    // Motor axes
    {attribute 'pytmc' := 'pv: CRIX:DPL:MMS:X'}
    {attribute 'TcLinkTo' := '.bLimitForwardEnable  := TIID^Device 1 (EtherCAT)^Term 5 (EK1200)^Term 6 (EK1122-0080)^DRL02-EK0 (EK1101-0080)^DRL02-E1 (EL7031)^STM Status^Status^Digital input 2;
                              .bLimitBackwardEnable := TIID^Device 1 (EtherCAT)^Term 5 (EK1200)^Term 6 (EK1122-0080)^DRL02-EK0 (EK1101-0080)^DRL02-E1 (EL7031)^STM Status^Status^Digital input 1'}
    M1 : DUT_MotionStage := (bPowerSelf:=TRUE, nEnableMode:=ENUM_StageEnableMode.DURING_MOTION);
    //stDPXMotor : DUT_MotionStage;

    {attribute 'pytmc' := 'pv: CRIX:DPL:MMS:Y'}
    {attribute 'TcLinkTo' := '.bLimitForwardEnable  := TIID^Device 1 (EtherCAT)^Term 5 (EK1200)^Term 6 (EK1122-0080)^DRL02-EK0 (EK1101-0080)^DRL02-E3 (EL7031)^STM Status^Status^Digital input 1;
                              .bLimitBackwardEnable := TIID^Device 1 (EtherCAT)^Term 5 (EK1200)^Term 6 (EK1122-0080)^DRL02-EK0 (EK1101-0080)^DRL02-E3 (EL7031)^STM Status^Status^Digital input 2'}
    M2 : DUT_MotionStage := (bPowerSelf:=TRUE, nEnableMode:=ENUM_StageEnableMode.DURING_MOTION);
    //stDPYMotor : DUT_MotionStage;

    {attribute 'pytmc' := 'pv: CRIX:DPL:MMS:Z'}
    {attribute 'TcLinkTo' := '.bLimitForwardEnable  := TIID^Device 1 (EtherCAT)^Term 5 (EK1200)^Term 6 (EK1122-0080)^DRL02-EK0 (EK1101-0080)^DRL02-E4 (EL7031)^STM Status^Status^Digital input 1;
                              .bLimitBackwardEnable := TIID^Device 1 (EtherCAT)^Term 5 (EK1200)^Term 6 (EK1122-0080)^DRL02-EK0 (EK1101-0080)^DRL02-E4 (EL7031)^STM Status^Status^Digital input 2'}
    M3 : DUT_MotionStage :=(bPowerSelf:=TRUE,nEnableMode:=ENUM_StageEnableMode.DURING_MOTION);
    //stDPZMotor : DUT_MotionStage;




    {attribute 'pytmc' := 'pv: CRIX:OBJ:MMS:X'}
    {attribute 'TcLinkTo' := '.bLimitForwardEnable  := TIID^Device 1 (EtherCAT)^Term 5 (EK1200)^Term 6 (EK1122-0080)^DRL02-EK0 (EK1101-0080)^DRL02-E6 (EL7031)^STM Status^Status^Digital input 2;
                              .bLimitBackwardEnable := TIID^Device 1 (EtherCAT)^Term 5 (EK1200)^Term 6 (EK1122-0080)^DRL02-EK0 (EK1101-0080)^DRL02-E6 (EL7031)^STM Status^Status^Digital input 1'}
    M4: DUT_MotionStage :=(bPowerSelf:=TRUE ,nEnableMode:=ENUM_StageEnableMode.DURING_MOTION);
    //stOBJXMotor : DUT_MotionStage;

    {attribute 'pytmc' := 'pv: CRIX:OBJ:MMS:Y'}
    {attribute 'TcLinkTo' := '.bLimitForwardEnable  := TIID^Device 1 (EtherCAT)^Term 5 (EK1200)^Term 6 (EK1122-0080)^DRL02-EK0 (EK1101-0080)^DRL02-E7 (EL7031)^STM Status^Status^Digital input 1;
                              .bLimitBackwardEnable := TIID^Device 1 (EtherCAT)^Term 5 (EK1200)^Term 6 (EK1122-0080)^DRL02-EK0 (EK1101-0080)^DRL02-E7 (EL7031)^STM Status^Status^Digital input 2'}
    M5 : DUT_MotionStage :=(bPowerSelf:=TRUE, nEnableMode:=ENUM_StageEnableMode.DURING_MOTION);
    //stOBJYMotor : DUT_MotionStage;

    {attribute 'pytmc' := 'pv: CRIX:OBJ:MMS:Z'}
    {attribute 'TcLinkTo' := '.bLimitForwardEnable  := TIID^Device 1 (EtherCAT)^Term 5 (EK1200)^Term 6 (EK1122-0080)^DRL02-EK0 (EK1101-0080)^DRL02-E9 (EL7031)^STM Status^Status^Digital input 1;
                              .bLimitBackwardEnable := TIID^Device 1 (EtherCAT)^Term 5 (EK1200)^Term 6 (EK1122-0080)^DRL02-EK0 (EK1101-0080)^DRL02-E9 (EL7031)^STM Status^Status^Digital input 2'}
    M6 : DUT_MotionStage :=(bPowerSelf:=TRUE, nEnableMode:=ENUM_StageEnableMode.DURING_MOTION);
    //stOBJZMotor : DUT_MotionStage;



    {attribute 'pytmc' := 'pv: CRIX:PDET:MMS:Y'}
    {attribute 'TcLinkTo' := '.bLimitForwardEnable  := TIID^Device 1 (EtherCAT)^Term 5 (EK1200)^Term 6 (EK1122-0080)^DRL02-EK0 (EK1101-0080)^DRL02-E11 (EL7031)^STM Status^Status^Digital input 1;
                              .bLimitBackwardEnable := TIID^Device 1 (EtherCAT)^Term 5 (EK1200)^Term 6 (EK1122-0080)^DRL02-EK0 (EK1101-0080)^DRL02-E11 (EL7031)^STM Status^Status^Digital input 2'}
    M7 : DUT_MotionStage := (bPowerSelf:=TRUE, nEnableMode:=ENUM_StageEnableMode.DURING_MOTION);
    //stPDYMotor : DUT_MotionStage;
    {attribute 'pytmc' := 'pv: CRIX:PDET:MMS:THETA'}
    {attribute 'TcLinkTo' := '.bLimitForwardEnable  := TIID^Device 1 (EtherCAT)^Term 5 (EK1200)^Term 6 (EK1122-0080)^DRL02-EK0 (EK1101-0080)^DRL02-E13 (EL7041)^STM Status^Status^Digital input 1;
                              .bLimitBackwardEnable := TIID^Device 1 (EtherCAT)^Term 5 (EK1200)^Term 6 (EK1122-0080)^DRL02-EK0 (EK1101-0080)^DRL02-E13 (EL7041)^STM Status^Status^Digital input 2'}
    M8 : DUT_MotionStage := (bPowerSelf:=TRUE, nEnableMode:=ENUM_StageEnableMode.DURING_MOTION);
    //stPDRotMotor : DUT_MotionStage;

    {attribute 'pytmc' := 'pv: CRIX:ILM:MMS:X'}
    {attribute 'TcLinkTo' := '.bLimitForwardEnable  := TIID^Device 1 (EtherCAT)^Term 5 (EK1200)^Term 6 (EK1122-0080)^DRL02-EK0 (EK1101-0080)^Term 65 (EL1084)^Channel 1^Input;
                              .bLimitBackwardEnable := TIID^Device 1 (EtherCAT)^Term 5 (EK1200)^Term 6 (EK1122-0080)^DRL02-EK0 (EK1101-0080)^Term 65 (EL1084)^Channel 2^Input'}
    M9 : DUT_MotionStage := (bPowerSelf:=TRUE, nEnableMode:=ENUM_StageEnableMode.DURING_MOTION); //stILMXMotor : DUT_MotionStage;

    {attribute 'pytmc' := 'pv: CRIX:ILM:MMS:Y'}
    {attribute 'TcLinkTo' := '.bLimitForwardEnable  := TIID^Device 1 (EtherCAT)^Term 5 (EK1200)^Term 6 (EK1122-0080)^DRL02-EK0 (EK1101-0080)^Term 65 (EL1084)^Channel 3^Input;
                              .bLimitBackwardEnable := TIID^Device 1 (EtherCAT)^Term 5 (EK1200)^Term 6 (EK1122-0080)^DRL02-EK0 (EK1101-0080)^Term 65 (EL1084)^Channel 4^Input'}
    M10 : DUT_MotionStage := (bPowerSelf:=TRUE, nEnableMode:=ENUM_StageEnableMode.DURING_MOTION); //stILMYMotor : DUT_MotionStage;

    {attribute 'pytmc' := 'pv: CRIX:ILM:MMS:Z'}
    {attribute 'TcLinkTo' := '.bLimitForwardEnable  := TIID^Device 1 (EtherCAT)^Term 5 (EK1200)^Term 6 (EK1122-0080)^DRL02-EK0 (EK1101-0080)^Term 68 (EL1084)^Channel 1^Input;
                              .bLimitBackwardEnable := TIID^Device 1 (EtherCAT)^Term 5 (EK1200)^Term 6 (EK1122-0080)^DRL02-EK0 (EK1101-0080)^Term 68 (EL1084)^Channel 2^Input'}
    M11 : DUT_MotionStage := (bPowerSelf:=TRUE, nEnableMode:=ENUM_StageEnableMode.DURING_MOTION); //stILMZMotor : DUT_MotionStage;

    {attribute 'pytmc' := 'pv: CRIX:QSTR:MMS:X'}
    {attribute 'TcLinkTo' := '.bLimitForwardEnable  := TIID^Device 1 (EtherCAT)^Term 5 (EK1200)^Term 6 (EK1122-0080)^DRL02-EK0 (EK1101-0080)^DRL02-E17 (EL7031)^STM Status^Status^Digital input 1;
                              .bLimitBackwardEnable := TIID^Device 1 (EtherCAT)^Term 5 (EK1200)^Term 6 (EK1122-0080)^DRL02-EK0 (EK1101-0080)^DRL02-E17 (EL7031)^STM Status^Status^Digital input 2'}
    M12 : DUT_MotionStage := (bPowerSelf:=TRUE, nEnableMode:=ENUM_StageEnableMode.DURING_MOTION);
    //stQSTXMotor : DUT_MotionStage;
    {attribute 'pytmc' := 'pv: CRIX:QSTR:MMS:Y'}
    {attribute 'TcLinkTo' := '.bLimitForwardEnable  := TIID^Device 1 (EtherCAT)^Term 5 (EK1200)^Term 6 (EK1122-0080)^DRL02-EK0 (EK1101-0080)^DRL02-E19 (EL7031)^STM Status^Status^Digital input 1;
                              .bLimitBackwardEnable := TIID^Device 1 (EtherCAT)^Term 5 (EK1200)^Term 6 (EK1122-0080)^DRL02-EK0 (EK1101-0080)^DRL02-E19 (EL7031)^STM Status^Status^Digital input 2'}
    M13 : DUT_MotionStage := (bPowerSelf:=TRUE, nEnableMode:=ENUM_StageEnableMode.DURING_MOTION);
    //stQSTYMotor : DUT_MotionStage;

    M14 : DUT_MotionStage; // SPARE 1
    M15 : DUT_MotionStage; // SPARE 2

    {attribute 'pytmc' := 'pv: CRIX:SDS:MMS:X'}
    M16 : DUT_MotionStage := (bPowerSelf:=TRUE, nEnableMode:=ENUM_StageEnableMode.DURING_MOTION); //stSDSXMotor : DUT_MotionStage;

    {attribute 'pytmc' := 'pv: CRIX:SDS:MMS:Y'}
    {attribute 'TcLinkTo' := '.bLimitForwardEnable := TIID^Device 1 (EtherCAT)^Term 5 (EK1200)^Term 6 (EK1122-0080)^DRL02-EK0 (EK1101-0080)^DRL02-E26 (EL7031)^STM Status^Status^Digital input 1;
                              .bLimitBackwardEnable := TIID^Device 1 (EtherCAT)^Term 5 (EK1200)^Term 6 (EK1122-0080)^DRL02-EK0 (EK1101-0080)^DRL02-E26 (EL7031)^STM Status^Status^Digital input 2'}
    M17 : DUT_MotionStage := (bPowerSelf:=TRUE, nEnableMode:=ENUM_StageEnableMode.DURING_MOTION); //stSDSYMotor : DUT_MotionStage;

    {attribute 'pytmc' := 'pv: CRIX:SDS:MMS:Z'}
    {attribute 'TcLinkTo' := '.bLimitForwardEnable := TIID^Device 1 (EtherCAT)^Term 5 (EK1200)^Term 6 (EK1122-0080)^DRL02-EK0 (EK1101-0080)^DRL02-E27 (EL7031)^STM Status^Status^Digital input 1'}
    M18 : DUT_MotionStage := (bPowerSelf:=TRUE, nEnableMode:=ENUM_StageEnableMode.DURING_MOTION); //stSDSZMotor : DUT_MotionStage;

    {attribute 'pytmc' := 'pv: CRIX:SDS:MMS:RX'}
(*	{attribute 'TcLinkTo' := '.bLimitForwardEnable := ;   // There are currently no limits on this stage
                              .bLimitBackwardEnable := '} *)
    M19 : DUT_MotionStage := (bPowerSelf:=TRUE, nEnableMode:=ENUM_StageEnableMode.DURING_MOTION); //stSDSRotMotor : DUT_MotionStage;

    {attribute 'pytmc' := 'pv: CRIX:SDS:MMS:RJET'}
(*	{attribute 'TcLinkTo' := '.bLimitForwardEnable := ;  // There are currently no limits on this stage
                              .bLimitBackwardEnable := '} *)
    M20 : DUT_MotionStage := (bPowerSelf:=TRUE, nEnableMode:=ENUM_StageEnableMode.DURING_MOTION); //stSDSShroudMotor : DUT_MotionStage;

    {attribute 'pytmc' := 'pv: CRIX:SDS:MMS:ZENCODER'}
    M36 : DUT_MotionStage; // SDS Z Encoder Axis

    {attribute 'pytmc' := 'pv: CRIX:CRYO:MMS:X'}
    {attribute 'TcLinkTo' := '.bLimitForwardEnable  := TIID^Device 1 (EtherCAT)^Term 5 (EK1200)^Term 6 (EK1122-0080)^DRL02-EK0 (EK1101-0080)^DRL02-ECJ1 (EK1122)^CryoStat (EK1101)^Cryo X (EL7041)^STM Status^Status^Digital input 1;
                              .bLimitBackwardEnable := TIID^Device 1 (EtherCAT)^Term 5 (EK1200)^Term 6 (EK1122-0080)^DRL02-EK0 (EK1101-0080)^DRL02-ECJ1 (EK1122)^CryoStat (EK1101)^Cryo X (EL7041)^STM Status^Status^Digital input 2'}
    M22 : DUT_MotionStage := (bPowerSelf:=TRUE, nEnableMode:=ENUM_StageEnableMode.DURING_MOTION); //CryoStat X
    {attribute 'pytmc' := 'pv: CRIX:CRYO:MMS:Y'}
    {attribute 'TcLinkTo' := '.bLimitForwardEnable  := TIID^Device 1 (EtherCAT)^Term 5 (EK1200)^Term 6 (EK1122-0080)^DRL02-EK0 (EK1101-0080)^DRL02-ECJ1 (EK1122)^CryoStat (EK1101)^Cryo Y (EL7041)^STM Status^Status^Digital input 1;
                              .bLimitBackwardEnable := TIID^Device 1 (EtherCAT)^Term 5 (EK1200)^Term 6 (EK1122-0080)^DRL02-EK0 (EK1101-0080)^DRL02-ECJ1 (EK1122)^CryoStat (EK1101)^Cryo Y (EL7041)^STM Status^Status^Digital input 2'}
    M23 : DUT_MotionStage := (bPowerSelf:=TRUE, nEnableMode:=ENUM_StageEnableMode.DURING_MOTION); //CryoStat Y
    {attribute 'pytmc' := 'pv: CRIX:CRYO:MMS:Z'}
    {attribute 'TcLinkTo' := '.bLimitForwardEnable  := TIID^Device 1 (EtherCAT)^Term 5 (EK1200)^Term 6 (EK1122-0080)^DRL02-EK0 (EK1101-0080)^DRL02-ECJ1 (EK1122)^CryoStat (EK1101)^Cryo Z (EL7041)^STM Status^Status^Digital input 1;
                              .bLimitBackwardEnable := TIID^Device 1 (EtherCAT)^Term 5 (EK1200)^Term 6 (EK1122-0080)^DRL02-EK0 (EK1101-0080)^DRL02-ECJ1 (EK1122)^CryoStat (EK1101)^Cryo Z (EL7041)^STM Status^Status^Digital input 2'}
    M24 : DUT_MotionStage:= (bPowerSelf:=TRUE, nEnableMode:=ENUM_StageEnableMode.DURING_MOTION); //CryoStat Z
    {attribute 'pytmc' := 'pv: CRIX:CRYO:MMS:RY'}
    M25 : DUT_MotionStage := (bPowerSelf:=TRUE, nEnableMode:=ENUM_StageEnableMode.DURING_MOTION); //CryoStat rY
     {attribute 'pytmc' := 'pv: CRIX:RCI:MMS:X'}
     {attribute 'TcLinkTo' := '.bLimitForwardEnable  := TIID^Device 1 (EtherCAT)^Term 5 (EK1200)^Term 6 (EK1122-0080)^DRL02-EK0 (EK1101-0080)^DRL02-ECJ0 (EK1122-0080)^RCI (EK1101-0080)^RCI X (EL7041)^STM Status^Status^Digital input 1;
                              .bLimitBackwardEnable := TIID^Device 1 (EtherCAT)^Term 5 (EK1200)^Term 6 (EK1122-0080)^DRL02-EK0 (EK1101-0080)^DRL02-ECJ0 (EK1122-0080)^RCI (EK1101-0080)^RCI X (EL7041)^STM Status^Status^Digital input 2'}
    M26 : DUT_MotionStage := (bPowerSelf:=TRUE, nEnableMode:=ENUM_StageEnableMode.DURING_MOTION); //RCI X
     {attribute 'pytmc' := 'pv: CRIX:RCI:MMS:Y'}
     {attribute 'TcLinkTo' := '.bLimitForwardEnable  := TIID^Device 1 (EtherCAT)^Term 5 (EK1200)^Term 6 (EK1122-0080)^DRL02-EK0 (EK1101-0080)^DRL02-ECJ0 (EK1122-0080)^RCI (EK1101-0080)^RCI Y (EL7041)^STM Status^Status^Digital input 1;
                              .bLimitBackwardEnable := TIID^Device 1 (EtherCAT)^Term 5 (EK1200)^Term 6 (EK1122-0080)^DRL02-EK0 (EK1101-0080)^DRL02-ECJ0 (EK1122-0080)^RCI (EK1101-0080)^RCI Y (EL7041)^STM Status^Status^Digital input 2'}
    M27 : DUT_MotionStage := (bPowerSelf:=TRUE, nEnableMode:=ENUM_StageEnableMode.DURING_MOTION); //RCI Y
     {attribute 'pytmc' := 'pv: CRIX:RCI:MMS:Z'}
     {attribute 'TcLinkTo' := '.bLimitForwardEnable  := TIID^Device 1 (EtherCAT)^Term 5 (EK1200)^Term 6 (EK1122-0080)^DRL02-EK0 (EK1101-0080)^DRL02-ECJ0 (EK1122-0080)^RCI (EK1101-0080)^RCI Z (EL7041)^STM Status^Status^Digital input 1;
                              .bLimitBackwardEnable := TIID^Device 1 (EtherCAT)^Term 5 (EK1200)^Term 6 (EK1122-0080)^DRL02-EK0 (EK1101-0080)^DRL02-ECJ0 (EK1122-0080)^RCI (EK1101-0080)^RCI Z (EL7041)^STM Status^Status^Digital input 2'}
    M28 : DUT_MotionStage := (bPowerSelf:=TRUE, nEnableMode:=ENUM_StageEnableMode.DURING_MOTION); //RCI Z
     {attribute 'pytmc' := 'pv: CRIX:RCI:MMS:RX'}
    M29 : DUT_MotionStage := (bPowerSelf:=TRUE, nEnableMode:=ENUM_StageEnableMode.DURING_MOTION); //RCI rX
     {attribute 'pytmc' := 'pv: CRIX:FZP:MMS:Y'}
     {attribute 'TcLinkTo' := '.bLimitForwardEnable  := TIID^Device 1 (EtherCAT)^Term 5 (EK1200)^Term 6 (EK1122-0080)^DRL02-EK0 (EK1101-0080)^DRL02-ECJ0 (EK1122-0080)^Term 113 (EK1101-0080)^FZP Y (EL7041)^STM Status^Status^Digital input 1;
                              .bLimitBackwardEnable := TIID^Device 1 (EtherCAT)^Term 5 (EK1200)^Term 6 (EK1122-0080)^DRL02-EK0 (EK1101-0080)^DRL02-ECJ0 (EK1122-0080)^Term 113 (EK1101-0080)^FZP Y (EL7041)^STM Status^Status^Digital input 2'}
    M30 : DUT_MotionStage := (bPowerSelf:=TRUE, nEnableMode:=ENUM_StageEnableMode.DURING_MOTION); //FZP Y
     {attribute 'pytmc' := 'pv: CRIX:FZP:MMS:X'}
     {attribute 'TcLinkTo' := '.bLimitForwardEnable  := TIID^Device 1 (EtherCAT)^Term 5 (EK1200)^Term 6 (EK1122-0080)^DRL02-EK0 (EK1101-0080)^DRL02-ECJ0 (EK1122-0080)^Term 113 (EK1101-0080)^FZP X (EL7041)^STM Status^Status^Digital input 1;
                              .bLimitBackwardEnable := TIID^Device 1 (EtherCAT)^Term 5 (EK1200)^Term 6 (EK1122-0080)^DRL02-EK0 (EK1101-0080)^DRL02-ECJ0 (EK1122-0080)^Term 113 (EK1101-0080)^FZP X (EL7041)^STM Status^Status^Digital input 2'}
    M31 : DUT_MotionStage := (bPowerSelf:=TRUE, nEnableMode:=ENUM_StageEnableMode.DURING_MOTION); //FZP X
     {attribute 'pytmc' := 'pv: CRIX:FZP:MMS:Z'}
     {attribute 'TcLinkTo' := '.bLimitForwardEnable  := TIID^Device 1 (EtherCAT)^Term 5 (EK1200)^Term 6 (EK1122-0080)^DRL02-EK0 (EK1101-0080)^DRL02-ECJ0 (EK1122-0080)^Term 113 (EK1101-0080)^FZP Z (EL7041)^STM Status^Status^Digital input 1;
                              .bLimitBackwardEnable := TIID^Device 1 (EtherCAT)^Term 5 (EK1200)^Term 6 (EK1122-0080)^DRL02-EK0 (EK1101-0080)^DRL02-ECJ0 (EK1122-0080)^Term 113 (EK1101-0080)^FZP Z (EL7041)^STM Status^Status^Digital input 2'}
    M32 : DUT_MotionStage := (bPowerSelf:=TRUE, nEnableMode:=ENUM_StageEnableMode.DURING_MOTION); //FZP Z
     {attribute 'pytmc' := 'pv: CRIX:CAM:MMS:X'}
     {attribute 'TcLinkTo' := '.bLimitForwardEnable  := TIID^Device 1 (EtherCAT)^Term 5 (EK1200)^Term 6 (EK1122-0080)^DRL02-EK0 (EK1101-0080)^DRL02-ECJ0 (EK1122-0080)^Term 109 (EK1101-0080)^Camera X (EL7041)^STM Status^Status^Digital input 1;
                              .bLimitBackwardEnable := TIID^Device 1 (EtherCAT)^Term 5 (EK1200)^Term 6 (EK1122-0080)^DRL02-EK0 (EK1101-0080)^DRL02-ECJ0 (EK1122-0080)^Term 109 (EK1101-0080)^Camera X (EL7041)^STM Status^Status^Digital input 2'}
    M33 : DUT_MotionStage := (bPowerSelf:=TRUE, nEnableMode:=ENUM_StageEnableMode.DURING_MOTION); //CAM X
     {attribute 'pytmc' := 'pv: CRIX:CAM:MMS:Y'}
     {attribute 'TcLinkTo' := '.bLimitForwardEnable  := TIID^Device 1 (EtherCAT)^Term 5 (EK1200)^Term 6 (EK1122-0080)^DRL02-EK0 (EK1101-0080)^DRL02-ECJ0 (EK1122-0080)^Term 109 (EK1101-0080)^Camera Y (EL7041)^STM Status^Status^Digital input 1;
                              .bLimitBackwardEnable := TIID^Device 1 (EtherCAT)^Term 5 (EK1200)^Term 6 (EK1122-0080)^DRL02-EK0 (EK1101-0080)^DRL02-ECJ0 (EK1122-0080)^Term 109 (EK1101-0080)^Camera Y (EL7041)^STM Status^Status^Digital input 2'}
    M34 : DUT_MotionStage := (bPowerSelf:=TRUE, nEnableMode:=ENUM_StageEnableMode.DURING_MOTION); //CAM Z
     {attribute 'pytmc' := 'pv: CRIX:OUTCOUP:MMS:Y'}
     {attribute 'TcLinkTo' := '.bLimitForwardEnable  := TIID^Device 1 (EtherCAT)^Term 5 (EK1200)^Term 6 (EK1122-0080)^DRL02-EK0 (EK1101-0080)^DRL02-E31 (EL7031)^STM Status^Status^Digital input 1;
                              .bLimitBackwardEnable := TIID^Device 1 (EtherCAT)^Term 5 (EK1200)^Term 6 (EK1122-0080)^DRL02-EK0 (EK1101-0080)^DRL02-E31 (EL7031)^STM Status^Status^Digital input 2'}
    M35 : DUT_MotionStage := (bPowerSelf:=TRUE, nEnableMode:=ENUM_StageEnableMode.DURING_MOTION); //OUTCOUP LENS Y

(*
    M21 : DUT_MotionStage; // Out-coupling y
 *)

 (* not needed for now; it has a manual knob
 // NOTE: Questar is M21, even though Outcoupling Y stage is before it on the DIN rail
     {attribute 'pytmc' := 'pv: CRIX:QSTR:MMS:FOCUS'}
    {attribute 'TcLinkTo' := '.bLimitForwardEnable  := TIID^Device 1 (EtherCAT)^Term 5 (EK1200)^Term 6 (EK1122-0080)^DRL02-EK0 (EK1101-0080)^DRL02-E33 (EL7031)^STM Status^Status^Digital input 1;
                              .bLimitBackwardEnable := TIID^Device 1 (EtherCAT)^Term 5 (EK1200)^Term 6 (EK1122-0080)^DRL02-EK0 (EK1101-0080)^DRL02-E33 (EL7031)^STM Status^Status^Digital input 2'}
    M21 : DUT_MotionStage; // Questar Focus
*)
    //Catcher Axes
     {attribute 'pytmc' := 'pv: CRIX:RCC:MMS:X'}
     {attribute 'TcLinkTo' := '.bLimitForwardEnable  := TIIB[Catcher_E1_EL7041]^STM Status^Status^Digital input 2;
                              .bLimitBackwardEnable := TIIB[Catcher_E1_EL7041]^STM Status^Status^Digital input 1'}
    M37 : DUT_MotionStage := (bPowerSelf:=TRUE, nEnableMode:=ENUM_StageEnableMode.DURING_MOTION); //RCC X
     {attribute 'pytmc' := 'pv: CRIX:RCC:MMS:Y'}
     {attribute 'TcLinkTo' := '.bLimitForwardEnable  := TIIB[Catcher_E3_EL7041]^STM Status^Status^Digital input 1;
                              .bLimitBackwardEnable := TIIB[Catcher_E3_EL7041]^STM Status^Status^Digital input 2'}
    M38 : DUT_MotionStage := (bPowerSelf:=TRUE, nEnableMode:=ENUM_StageEnableMode.DURING_MOTION); //RCC Y
     {attribute 'pytmc' := 'pv: CRIX:RCC:MMS:Z'}
     {attribute 'TcLinkTo' := '.bLimitForwardEnable  := TIIB[Catcher_E4_EL7041]^STM Status^Status^Digital input 2;
                              .bLimitBackwardEnable := TIIB[Catcher_E4_EL7041]^STM Status^Status^Digital input 1'}
    M39 : DUT_MotionStage := (bPowerSelf:=TRUE, nEnableMode:=ENUM_StageEnableMode.DURING_MOTION); //RCC Z

     // VLS SLIT TOP
    {attribute 'TcLinkTo' := '	.bLimitForwardEnable:=TIIB[VLS_EP6_EP7041-1002]^STM Status^Status^Digital input 1;
                                .bLimitBackwardEnable:=TIIB[VLS_EP6_EP7041-1002]^STM Status^Status^Digital input 2'}
    {attribute 'pytmc' := '
        pv: CRIX:VLS:MMS:SLTOP
        field: DESC VLS Slit TOP Blade
    '}
    M40: DUT_MotionStage;

     // VLS SLIT BOTTOM
    {attribute 'TcLinkTo' := '	.bLimitForwardEnable:=TIIB[VLS_EP7_EP7041-1002]^STM Status^Status^Digital input 1;
                                .bLimitBackwardEnable:=TIIB[VLS_EP7_EP7041-1002]^STM Status^Status^Digital input 2'}
    {attribute 'pytmc' := '
        pv: CRIX:VLS:MMS:SLBOTTOM
        field: DESC VLS Slit BOTTOM Blade
    '}
    M41: DUT_MotionStage;

    // VLS SLIT RIGHT
    {attribute 'TcLinkTo' := '	.bLimitForwardEnable:=TIIB[VLS_EP8_EP7041-1002]^STM Status^Status^Digital input 1;
                                .bLimitBackwardEnable:=TIIB[VLS_EP8_EP7041-1002]^STM Status^Status^Digital input 2'}
    {attribute 'pytmc' := '
        pv: CRIX:VLS:MMS:SLRIGHT
        field: DESC VLS Slit RIGHT Blade
    '}
    M42: DUT_MotionStage;


    // VLS SLIT LEFT
    {attribute 'TcLinkTo' := '	.bLimitForwardEnable:=TIIB[VLS_EP9_EP7041-1002]^STM Status^Status^Digital input 1;
                                .bLimitBackwardEnable:=TIIB[VLS_EP9_EP7041-1002]^STM Status^Status^Digital input 2'}
    {attribute 'pytmc' := '
        pv: CRIX:VLS:MMS:SLLEFT
        field: DESC VLS Slit LEFT Blade
    '}
    M43: DUT_MotionStage;



    // VLS focusing mirror pitch
    {attribute 'TcLinkTo' := '	.bLimitForwardEnable:=TIIB[VLS_EP10_EP7041-3102]^STM Status^Status^Digital input 2;
                                .bLimitBackwardEnable:=TIIB[VLS_EP10_EP7041-3102]^STM Status^Status^Digital input 1;
                                .nRawEncoderUINT:=TIIB[VLS_EP10_EP7041-3102]^ENC Status compact^Counter value;
                                .bHome:=TIIB[VLS_EP10_EP7041-3102]^ENC Status compact^Status^Status of input C'}
    {attribute 'pytmc' := '
        pv:  CRIX:VLS:MMS:MP
        field: DESC VLS Focus Mirror
    '}
    M44: DUT_MotionStage;

    // VLS grating pitch
    {attribute 'TcLinkTo' := '	.bLimitForwardEnable:=TIIB[VLS_EP11_EP7041-3102]^STM Status^Status^Digital input 2;
                                .bLimitBackwardEnable:=TIIB[VLS_EP11_EP7041-3102]^STM Status^Status^Digital input 1;
                                .nRawEncoderUINT:=TIIB[VLS_EP11_EP7041-3102]^ENC Status compact^Counter value;
                                .bHome:=TIIB[VLS_EP11_EP7041-3102]^ENC Status compact^Status^Status of input C'}
    {attribute 'pytmc' := '
        pv:  CRIX:VLS:MMS:GP
        field: DESC VLS Grating
    '}
    M45: DUT_MotionStage;

    // VLS camera Pitch
    {attribute 'TcLinkTo' := '	.bLimitForwardEnable:=TIIB[VLS_EP12_EP7041-3102]^STM Status^Status^Digital input 1;
                                .bLimitBackwardEnable:=TIIB[VLS_EP12_EP7041-3102]^STM Status^Status^Digital input 2;
                                .bHome:=TIIB[VLS_EP12_EP7041-3102]^ENC Status compact^Status^Status of input C'}
    {attribute 'pytmc' := '
        pv:  CRIX:VLS:CAM:MMS:PITCH
        field: DESC VLS Camera Pitch
    '}
    M46: DUT_MotionStage;

    // VLS camera Distance
    {attribute 'TcLinkTo' := '	.bLimitForwardEnable:=TIIB[VLS_EP13_EP7041-3102]^STM Status^Status^Digital input 2;
                                .bLimitBackwardEnable:=TIIB[VLS_EP13_EP7041-3102]^STM Status^Status^Digital input 1;
                                .bHome:=TIIB[VLS_EP13_EP7041-3102]^ENC Status compact^Status^Status of input C'}
    {attribute 'pytmc' := '
        pv:  CRIX:VLS:CAM:MMS:DIST
        field: DESC VLS Camera Translation
    '}
    M47: DUT_MotionStage;

    //Cryo pump
    {attribute 'TcLinkTo' := '	.bLimitForwardEnable:=TIIB[DRL02-E23 (EL7041)]^STM Status^Status^Digital input 2'}
    {attribute 'pytmc' := '
        pv:  CRIX:PTC:Y:MMS:10
        field:Cryo Pump Y stage 10
    '}
    M48: DUT_MotionStage;
    {attribute 'TcLinkTo' := '	.bLimitForwardEnable:=TIIB[DRL02-E21 (EL7041)]^STM Status^Status^Digital input 2'}
    {attribute 'pytmc' := '
        pv:  CRIX:PTC:Y:MMS:11
        field:Cryo Pump Y stage 11
    '}
    M49: DUT_MotionStage;

    // SL2K2-SCATTER: 4 Axes
    {attribute 'pytmc' := 'pv: SL2K2:SCATTER:MMS:BOTTOM'}
    {attribute 'TcLinkTo' := '.bLimitForwardEnable  := TIIB[SL2K2-EL7031-E1]^STM Status^Status^Digital input 2;
                             .bLimitBackwardEnable := TIIB[SL2K2-EL7031-E1]^STM Status^Status^Digital input 1;
                              .nRawEncoderUINT      := TIIB[SL2K2-EL5101-E2]^ENC Status compact^Counter value'}
    M50: DUT_MotionStage := (sName := 'SL2K2:SCATTER:MMS:BOTTOM');
    {attribute 'pytmc' := 'pv: SL2K2:SCATTER:MMS:TOP'}
    {attribute 'TcLinkTo' := '.bLimitForwardEnable  := TIIB[SL2K2-EL7031-E3]^STM Status^Status^Digital input 2;
                              .bLimitBackwardEnable := TIIB[SL2K2-EL7031-E3]^STM Status^Status^Digital input 1;
                              .nRawEncoderUINT      := TIIB[SL2K2-EL5101-E4]^ENC Status compact^Counter value'}
    M51: DUT_MotionStage := (sName := 'SL2K2:SCATTER:MMS:TOP');
    {attribute 'pytmc' := 'pv: SL2K2:SCATTER:MMS:NORTH'}
    {attribute 'TcLinkTo' := '.bLimitForwardEnable  := TIIB[SL2K2-EL7031-E5]^STM Status^Status^Digital input 1;
                              .bLimitBackwardEnable := TIIB[SL2K2-EL7031-E5]^STM Status^Status^Digital input 2;
                              .nRawEncoderUINT      := TIIB[SL2K2-EL5101-E6]^ENC Status compact^Counter value'}
    M52: DUT_MotionStage := (sName := 'SL2K2:SCATTER:MMS:NORTH');
    {attribute 'pytmc' := 'pv: SL2K2:SCATTER:MMS:SOUTH'}
    {attribute 'TcLinkTo' := '.bLimitForwardEnable  := TIIB[SL2K2-EL7031-E7]^STM Status^Status^Digital input 1;
                              .bLimitBackwardEnable := TIIB[SL2K2-EL7031-E7]^STM Status^Status^Digital input 2;
                              .nRawEncoderUINT      := TIIB[SL2K2-EL5101-E8]^ENC Status compact^Counter value'}
    M53: DUT_MotionStage := (sName := 'SL2K2:SCATTER:MMS:SOUTH');

END_VAR

// ---- POUs/Assemblies/PRG_FZP.TcPOU
PROGRAM PRG_FZP
VAR
    fbFZP_Motor_X : FB_MotionStage;
    fbFZP_Motor_Y : FB_MotionStage;
    fbFZP_Motor_Z : FB_MotionStage;
    fbOUTCOUP_Motor_Y : FB_MotionStage;
END_VAR

Main.M30.bHardwareEnable := TRUE;
fbFZP_Motor_Y(stMotionStage:=Main.M30);

Main.M31.bHardwareEnable := TRUE;
fbFZP_Motor_X(stMotionStage:=Main.M31);

Main.M32.bHardwareEnable := TRUE;
fbFZP_Motor_Z(stMotionStage:=Main.M32);

Main.M35.bHardwareEnable := TRUE;
fbOUTCOUP_Motor_Y(stMotionStage:=Main.M35);

END_PROGRAM

// ---- POUs/Assemblies/PRG_CryoPump.TcPOU
PROGRAM PRG_CryoPump
VAR
    fbCryoPump_Motor_Y_10 : FB_MotionStage;
    fbCryoPump_Motor_Y_11 : FB_MotionStage;

    bEPS_OK_Y_10: BOOL; //Valve is in the Open State And communication ok
    bEPS_OK_Y_11: BOOL; //Valve is in the Open State And communication ok

    bInit : BOOl := TRUE;

    (*Limit switches*)
    {attribute 'TcLinkTo' := 'TIIB[DRL02-E23 (EL7041)]^STM Status^Status^Digital input 1'}
    bLimitBackwardEnable_Y_10 AT %I* :BOOL;
    {attribute 'TcLinkTo' := 'TIIB[DRL02-E21 (EL7041)]^STM Status^Status^Digital input 1'}
    bLimitBackwardEnable_Y_11 AT %I* :BOOL;

    (*ETHERCAT BRRIDGE COM STATUS*)
    //0: Other side is in OP state, >0: Error
    {attribute 'pytmc' := 'pv:  CRIX:MOT2VAC:ECATBRG:TxPDO_state'}
    {attribute 'TcLinkTo' := 'TIIB[CRIX_VAC_INTF (EL6695-0002)]^SYNC Inputs^TxPDO state'}
    xEcatBridge_TxPDO_state AT %I* :BOOL;

    //0: External device connectd, 1: External device not connected
    {attribute 'pytmc' := 'pv:  CRIX:MOT2VAC:ECATBRG:External_device_not_connected'}
    {attribute 'TcLinkTo':= 'TIIB[CRIX_VAC_INTF (EL6695-0002)]^SYNC Inputs^External device not connected'}
    xEcatBridge_External_device_not_connected AT %I* : BOOL;

    //0 = Data valid, 1 = Data invalid
    {attribute 'pytmc' := 'pv:  CRIX:MOT2VAC:ECATBRG:WcState'}
    {attribute 'TcLinkTo' := 'TIIB[CRIX_VAC_INTF (EL6695-0002)]^WcState^WcState'}
    xEcatBridge_WcState AT %I* : BOOL;

    //Inputs
    {attribute 'TcLinkTo' := 'TIIB[CRIX_VAC_INTF (EL6695-0002)]^IO Inputs^bCRYO_VGC_01_CLS'}
    bCRYO_VGC_01_CLS AT %I* : BOOL;
    {attribute 'TcLinkTo' := 'TIIB[CRIX_VAC_INTF (EL6695-0002)]^IO Inputs^bCRYO_VGC_01_OPN'}
    bCRYO_VGC_01_OPN AT %I* : BOOL;
    {attribute 'TcLinkTo' := 'TIIB[CRIX_VAC_INTF (EL6695-0002)]^IO Inputs^bCRYO_VGC_02_CLS'}
    bCRYO_VGC_02_CLS AT %I* : BOOL;
    {attribute 'TcLinkTo' := 'TIIB[CRIX_VAC_INTF (EL6695-0002)]^IO Inputs^bCRYO_VGC_02_OPN'}
    bCRYO_VGC_02_OPN AT %I* : BOOL;

    //Outputs
    {attribute 'TcLinkTo' := 'TIIB[CRIX_VAC_INTF (EL6695-0002)]^IO Outputs^bMOTY10_IN'}
    bMOTY10_IN AT %Q* : BOOL;
    {attribute 'TcLinkTo' := 'TIIB[CRIX_VAC_INTF (EL6695-0002)]^IO Outputs^bMOTY10_OUT'}
    bMOTY10_OUT AT %Q* : BOOL;
    {attribute 'TcLinkTo' := 'TIIB[CRIX_VAC_INTF (EL6695-0002)]^IO Outputs^bMOTY11_IN'}
    bMOTY11_IN AT %Q* : BOOL;
    {attribute 'TcLinkTo' := 'TIIB[CRIX_VAC_INTF (EL6695-0002)]^IO Outputs^bMOTY11_OUT'}
    bMOTY11_OUT AT %Q* : BOOL;

END_VAR

IF ( bInit) THEN
    bInit := FALSE;
    Main.M48.bHardwareEnable := TRUE; //Linked to valve state
    Main.M48.bPowerSelf := TRUE;
    Main.M48.nBrakeMode := ENUM_StageBrakeMode.NO_BRAKE;
    Main.M48.nEnableMode := ENUM_StageEnableMode.DURING_MOTION;
    Main.M49.bHardwareEnable := TRUE; //Linked to valve state
    Main.M49.bPowerSelf := TRUE;
    Main.M49.nBrakeMode := ENUM_StageBrakeMode.NO_BRAKE;
    Main.M49.nEnableMode := ENUM_StageEnableMode.DURING_MOTION;

    //Homing routine parameters
    Main.M48.fHomePosition:= 0;
    Main.M48.nHomingMode := ENUM_EpicsHomeCmd.HIGH_LIMIT;
    Main.M49.fHomePosition:= 0;
    Main.M49.nHomingMode := ENUM_EpicsHomeCmd.HIGH_LIMIT;
END_IF

fbCryoPump_Motor_Y_10(stMotionStage:=Main.M48);
fbCryoPump_Motor_Y_11(stMotionStage:=Main.M49);

//Interface
bMOTY10_IN := NOT bLimitBackwardEnable_Y_10;
bMOTY10_OUT := NOT Main.M48.bLimitForwardEnable;
bMOTY11_IN := NOT bLimitBackwardEnable_Y_11;
bMOTY11_OUT := NOT Main.M49.bLimitForwardEnable;
bEPS_OK_Y_10 := (NOT bCRYO_VGC_01_CLS) AND bCRYO_VGC_01_OPN AND NOT (xEcatBridge_External_device_not_connected) AND NOT (xEcatBridge_WcState) AND NOT (xEcatBridge_TxPDO_state);
bEPS_OK_Y_11 := (NOT bCRYO_VGC_02_CLS) AND bCRYO_VGC_02_OPN AND NOT (xEcatBridge_External_device_not_connected) AND NOT (xEcatBridge_WcState) AND NOT (xEcatBridge_TxPDO_state);



//Handle EPS
Main.M48.bLimitBackwardEnable := bEPS_OK_Y_10 AND bLimitBackwardEnable_Y_10;
Main.M49.bLimitBackwardEnable := bEPS_OK_Y_11 AND bLimitBackwardEnable_Y_11;

END_PROGRAM

// ---- POUs/Assemblies/PRG_FiberLite.TcPOU
PROGRAM PRG_FiberLite
VAR


END_VAR

// Set LED output scaling (Fiber-Lite)
bLedOutput1.iTermBits := 14;
bLedOutput1(fbSetIllPercent=>);

bLedOutput2.iTermBits := 14;
bLedOutput2();

bLedOutput3.iTermBits := 14;
bLedOutput3();

bLedOutput4.iTermBits := 14;
bLedOutput4();

END_PROGRAM

// ---- POUs/Assemblies/PRG_InjectorMotors.TcPOU
PROGRAM PRG_InjectorMotors
VAR
    fbSDSX_Motor : FB_MotionStage;
    fbSDSY_Motor : FB_MotionStage;
    fbSDSZ_Motor : FB_MotionStage;
    fbSDSRY_Motor : FB_MotionStage;
    fbSDSShroud_Motor : FB_MotionStage;
    fbSDSZEncoder: FB_MotionStage;

    bEPS_OK_SDSZ_18: BOOL; //Valve is in the Open State And communication ok

    bInit : BOOL := TRUE;

    //Limit Switch
    {attribute 'TcLinkTo' := 'TIID^Device 1 (EtherCAT)^Term 5 (EK1200)^Term 6 (EK1122-0080)^DRL02-EK0 (EK1101-0080)^DRL02-E27 (EL7031)^STM Status^Status^Digital input 2'}
    bLimitBackwardEnable_SDSZ_18 AT %I* : BOOL;

    {attribute 'TcLinkTo' := 'TIIB[CRIX_VAC_INTF (EL6695-0002)]^IO Inputs^bSDS_VGC_01_CLS'}
    bSDS_VGC_01_CLS AT %I* : BOOL;
    {attribute 'TcLinkTo' := 'TIIB[CRIX_VAC_INTF (EL6695-0002)]^IO Inputs^bSDS_VGC_01_OPN'}
    bSDS_VGC_01_OPN AT %I* : BOOL;

    {attribute 'TcLinkTo' := 'TIIB[CRIX_VAC_INTF (EL6695-0002)]^IO Outputs^bMOTSDSZ18_IN'}
    bMOTSDSZ18_IN AT %Q* : BOOL;
    {attribute 'TcLinkTo' := 'TIIB[CRIX_VAC_INTF (EL6695-0002)]^IO Outputs^bMOTSDSZ18_OUT'}
    bMOTSDSZ18_OUT AT %Q* : BOOL;

    // Hall Effect Limits for SDS X Stage
    {attribute 'TcLinkTo' := 'TIID^Device 1 (EtherCAT)^Term 5 (EK1200)^Term 6 (EK1122-0080)^DRL02-EK0 (EK1101-0080)^Term 173 (EL1124)^Channel 3^Input'}
    bHall_Forward AT %I* : BOOL;
    nHall_Forward_Cycles: UINT;
    {attribute 'TcLinkTo' := 'TIID^Device 1 (EtherCAT)^Term 5 (EK1200)^Term 6 (EK1122-0080)^DRL02-EK0 (EK1101-0080)^Term 173 (EL1124)^Channel 4^Input'}
    bHall_Backward AT %I*: BOOL;
    nHall_Backward_Cycles: UINT;

    nNumCyclesNeeded: UINT := 10;

END_VAR

if (bInit) THEN
    // X Motor
    Main.M16.bHardwareEnable := TRUE;
    Main.M16.nHomingMode := ENUM_EpicsHomeCmd.ABSOLUTE_SET;
    // Y motor
    Main.M17.bHardwareEnable := TRUE;
    // Z Motor
    Main.M18.bHardwareEnable := TRUE;
    // Y Rotation Motor
    Main.M19.bHardwareEnable := TRUE;
    Main.M19.bLimitForwardEnable := TRUE;
    Main.M19.bLimitBackwardEnable := TRUE;
    // Shroud Motor
    Main.M20.bHardwareEnable := TRUE;
    Main.M20.bLimitForwardEnable := TRUE;
    Main.M20.bLimitBackwardEnable := TRUE;
END_IF

fbSDSX_Motor(stMotionStage:=Main.M16);
fbSDSY_Motor(stMotionStage:=Main.M17);
fbSDSZ_Motor(stMotionStage:=Main.M18);
fbSDSRY_Motor(stMotionStage:=Main.M19);
fbSDSShroud_Motor(stMotionStage:=Main.M20);
fbSDSZEncoder(stMotionStage:=Main.M36);


bMOTSDSZ18_OUT := NOT Main.M18.bLimitForwardEnable;
bMOTSDSZ18_IN := NOT bLimitBackwardEnable_SDSZ_18;
bEPS_OK_SDSZ_18 := (NOT bSDS_VGC_01_CLS) AND bSDS_VGC_01_OPN AND NOT (PRG_CryoPump.xEcatBridge_External_device_not_connected) AND NOT (PRG_CryoPump.xEcatBridge_WcState) AND NOT (PRG_CryoPump.xEcatBridge_TxPDO_state);


Main.M18.bLimitBackwardEnable := bEPS_OK_SDSZ_18 AND bLimitBackwardEnable_SDSZ_18;

// X Stage Groundswitching Limits Logic

//Cycle counting code for dealing with interference
IF bHall_Forward THEN
    nHall_Forward_Cycles := MIN(nHall_Forward_Cycles + 1, nNumCyclesNeeded);
ELSE
    nHall_Forward_Cycles := 0;
END_IF
IF bHall_Backward THEN
    nHall_Backward_Cycles := MIN(nHall_Backward_Cycles + 1, nNumCyclesNeeded);
ELSE
    nHall_Backward_Cycles := 0;
END_IF

Main.M16.bLimitForwardEnable := nHall_Forward_Cycles < nNumCyclesNeeded;
Main.M16.bLimitBackwardEnable := nHall_Backward_Cycles < nNumCyclesNeeded;

END_PROGRAM

// ---- POUs/Assemblies/PRG_VLS.TcPOU
PROGRAM PRG_VLS
VAR
    fbVLS_SLITS_TOP : FB_MotionStage;
    fbVLS_SLITS_BOTTOM : FB_MotionStage;
    fbVLS_SLITS_RIGHT : FB_MotionStage;
    fbVLS_SLITS_LEFT: FB_MotionStage;
    fbVLS_Mirror_P : FB_MotionStage;
    fbVLS_Grating_P : FB_MotionStage;
    fbVLS_CAM_P : FB_MotionStage;
    fbVLS_CAM_D : FB_MotionStage;

    bInit :BOOL:=TRUE;


    rGrating_Pitch :LREAL;
    rMirror_Pitch :LREAL;

END_VAR

IF ( bInit) THEN
    bInit := FALSE;
    //SLITS
    Main.M40.bHardwareEnable := TRUE;
    Main.M40.bPowerSelf :=TRUE;
    Main.M40.nBrakeMode := ENUM_StageBrakeMode.NO_BRAKE;
    Main.M40.nEnableMode := ENUM_StageEnableMode.DURING_MOTION;
    Main.M41.bHardwareEnable := TRUE;
    Main.M41.bPowerSelf :=TRUE;
    Main.M41.nBrakeMode := ENUM_StageBrakeMode.NO_BRAKE;
    Main.M41.nEnableMode := ENUM_StageEnableMode.DURING_MOTION;
    Main.M42.bHardwareEnable := TRUE;
    Main.M42.bPowerSelf :=TRUE;
    Main.M42.nBrakeMode := ENUM_StageBrakeMode.NO_BRAKE;
    Main.M42.nEnableMode := ENUM_StageEnableMode.DURING_MOTION;
    Main.M43.bHardwareEnable := TRUE;
    Main.M43.bPowerSelf :=TRUE;
    Main.M43.nBrakeMode := ENUM_StageBrakeMode.NO_BRAKE;
    Main.M43.nEnableMode := ENUM_StageEnableMode.DURING_MOTION;

    //Homing routine parameters
    Main.M40.fHomePosition:= 0;
    Main.M40.nHomingMode := ENUM_EpicsHomeCmd.LOW_LIMIT;
    Main.M41.fHomePosition:= 0;
    Main.M41.nHomingMode := ENUM_EpicsHomeCmd.LOW_LIMIT;
    Main.M42.fHomePosition:= 0;
    Main.M42.nHomingMode := ENUM_EpicsHomeCmd.LOW_LIMIT;
    Main.M43.fHomePosition:= 0;
    Main.M43.nHomingMode := ENUM_EpicsHomeCmd.LOW_LIMIT;

    //Focusing Mirror Pitch
    Main.M44.bHardwareEnable := TRUE;
    Main.M44.bPowerSelf :=TRUE;
    Main.M44.nBrakeMode := ENUM_StageBrakeMode.NO_BRAKE;
    Main.M44.nEnableMode := ENUM_StageEnableMode.DURING_MOTION;
    //Homing routine parameters
    Main.M44.fHomePosition:= -0.2288; // old homing position: -3.473;
    Main.M44.nHomingMode := ENUM_EpicsHomeCmd.LOW_LIMIT;

    //Grating Pitch
    Main.M45.bHardwareEnable := TRUE;
    Main.M45.bPowerSelf :=TRUE;
    Main.M45.nBrakeMode := ENUM_StageBrakeMode.NO_BRAKE;
    Main.M45.nEnableMode := ENUM_StageEnableMode.DURING_MOTION;
    //Homing routine parameters
    Main.M45.fHomePosition:= -1.74;
    Main.M45.nHomingMode := ENUM_EpicsHomeCmd.LOW_LIMIT;

    //Cam
    Main.M46.bHardwareEnable := TRUE;
    Main.M46.bPowerSelf :=TRUE;
    Main.M46.nBrakeMode := ENUM_StageBrakeMode.NO_BRAKE;
    Main.M46.nEnableMode := ENUM_StageEnableMode.DURING_MOTION;
    Main.M47.bHardwareEnable := TRUE;
    Main.M47.bPowerSelf :=TRUE;
    Main.M47.nBrakeMode := ENUM_StageBrakeMode.NO_BRAKE;
    Main.M47.nEnableMode := ENUM_StageEnableMode.DURING_MOTION;
    //Homing routine parameters
    Main.M46.fHomePosition:= 0.8923;
    Main.M46.nHomingMode := ENUM_EpicsHomeCmd.HIGH_LIMIT;//0 where it is horizontal
    Main.M47.fHomePosition:= -15.5;
    Main.M47.nHomingMode := ENUM_EpicsHomeCmd.LOW_LIMIT;
END_IF


//Calculate the mirror and grating pitch values
//OLD EQUATION:
//Mirror Pitch (x)  =   33.85 + 18.09x  - 0.2479x2
//rMirror_Pitch :=33.85 + (18.09*Main.M44.stAxisStatus.fActPosition(*mm*)  )- (0.2479 * EXPT(Main.M44.stAxisStatus.fActPosition,2));

//NEW EQUATION:
rMirror_Pitch :=27.667 + (18.1*Main.M44.stAxisStatus.fActPosition(*mm*)  )+ (-0.7569 * EXPT(Main.M44.stAxisStatus.fActPosition,2));

//Grating Pitch (x) =  22.56 - 16.25x + 0.334x2
rGrating_Pitch := 22.56 - (16.25*Main.M45.stAxisStatus.fActPosition(*mm*)  )+ (0.334 * EXPT(Main.M45.stAxisStatus.fActPosition,2));




fbVLS_SLITS_TOP(stMotionStage:=Main.M40);
fbVLS_SLITS_BOTTOM(stMotionStage:=Main.M41);
fbVLS_SLITS_RIGHT(stMotionStage:=Main.M42);
fbVLS_SLITS_LEFT(stMotionStage:=Main.M43);
fbVLS_Mirror_P(stMotionStage:=Main.M44);
fbVLS_Grating_P(stMotionStage:=Main.M45);
fbVLS_CAM_P(stMotionStage:=Main.M46);
fbVLS_CAM_D(stMotionStage:=Main.M47);

END_PROGRAM

// ---- POUs/EPS/InjectorMotorEPSLimits/FB_CheckEPS.TcPOU
FUNCTION_BLOCK FB_CheckEPS
VAR_IN_OUT
    stMotor	: ST_MotionStage;
    aEPSLimits : ARRAY [*] OF ST_EPSLimits;
    // Allows for user to define what is 'forward' and what is 'backward'. In most cases, use the in_out stMotor as default.
    stForwardMotorEPS : DUT_EPS;
    stBackwardMotorEPS: DUT_EPS;

END_VAR
VAR_INPUT
    // Encoder Position, Current position of motor. Needed for the case where the motor and encoders are seperate. Default use stMotor Position
    fPosition : LREAL;
    // Ignores EPS
    bEPS_Override : BOOL;

END_VAR
VAR_OUTPUT
END_VAR
VAR
    nPreviousState : DINT;
    nIndex: DINT;
    nEPSIndex: DINT;
    bUnknownState: BOOL;
    fbBwdEPS: FB_EPS;
    fbFwdEPS: FB_EPS;
END_VAR

fbBwdEps(eps:=stBackwardMotorEPS);
fbFwdEPS(eps:=stForwardMotorEPS);

// Look through possible states to see which state we are in
bUnknownState := TRUE;
FOR nIndex := LOWER_BOUND(aEPSLimits, 1) TO UPPER_BOUND(aEPSLimits, 1) BY 1 DO
    IF aEPSLimits[nIndex].stEPS.bEPS_OK THEN
        nEPSIndex := nIndex;
        bUnknownState := FALSE; // Known State
        exit; // stop when found state
    END_IF
END_FOR

IF (nPreviousState <> nEPSIndex) THEN
    // only clear stMotor eps from previous state.
    fbBwdEPS.setBit(DINT_TO_BYTE(0), TRUE);
    fbFwdEPS.setBit(DINT_TO_BYTE(0), TRUE);
END_IF

// Check if position is in plc limit rage, Stop motor if out of Upper/Lower bounds
IF fPosition > aEPSLimits[nEPSIndex].fBwd_Limits THEN
    fbBwdEPS.setBit(DINT_TO_BYTE(0), TRUE);
ELSE
    fbBwdEPS.setBit(DINT_TO_BYTE(0), FALSE);
END_IF

IF fPosition < aEPSLimits[nEPSIndex].fFwd_Limits THEN
    fbFwdEPS.setBit(DINT_TO_BYTE(0), TRUE);
ELSE
    fbFwdEPS.setBit(DINT_TO_BYTE(0), FALSE);
END_IF

IF bUnknownState THEN
    stBackwardMotorEPS.bEPS_OK := FALSE;
    stForwardMotorEPS.bEPS_OK := FALSE;

    stBackwardMotorEPS.sMessage := 'UNKNOWN STATE';
    stForwardMotorEPS.sMessage := 'UNKNOWN STATE';
    ELSE
    // Update Labels
    stBackwardMotorEPS.sMessage := aEPSLimits[nEPSIndex].stEPS.sMessage;
    stForwardMotorEPS.sMessage := aEPSLimits[nEPSIndex].stEPS.sMessage;
END_IF

IF bEPS_Override THEN
    stBackwardMotorEPS.bEPS_OK := TRUE;
    stForwardMotorEPS.bEPS_OK := TRUE;
END_IF

nPreviousState := nEPSIndex; // Update Previous State

END_FUNCTION_BLOCK

// ---- POUs/EPS/InjectorMotorEPSLimits/F_InRange.TcPOU
FUNCTION F_InRange : BOOL
// Determine if value is between the lower and upper limit
VAR_INPUT
    value 		: LREAL;
    lower_limit : LREAL;
    upper_limit : LREAL;
END_VAR
VAR
END_VAR

F_InRange := (lower_limit < value) AND (value < upper_limit);

END_FUNCTION

// ---- POUs/EPS/InjectorMotorEPSLimits/FB_RestTimer.TcPOU
FUNCTION_BLOCK FB_RestTimer
// Resets value of input after some time
// bInput 	: Value that will reset when set to true after some time passes
// tCountdown : count down when input will be rest
// tElapseTime : Time before input is reset

VAR_IN_OUT
    bInput : BOOL;
    tCountDown : STRING;
END_VAR
VAR_INPUT
    tElapseTime : TIME;
END_VAR
VAR
    fbTimer : TON;
END_VAR

fbTimer(IN := bInput, PT:= tElapseTime);

IF bInput THEN
    tCountDown := TIME_TO_STRING(tElapseTime - fbTimer.ET);
END_IF

IF fbTimer.Q THEN
    bInput := FALSE;
    tCountDown := TIME_TO_STRING(T#0s);
END_IF

END_FUNCTION_BLOCK

// ---- POUs/EPS/InjectorMotorEPSLimits/PRG_DPL_X_EPS.TcPOU
PROGRAM PRG_DPL_X_EPS
VAR
    {attribute 'pytmc' := 'pv: CRIX:DPL:MMS:X:EPS'}
    aDPL_X_EPS		: ARRAY [1 .. 3] OF ST_EPSLimits;

    {attribute 'pytmc' := 'pv: CRIX:DPL:MMS:X:EPS:OVRD_MODE'}
    bEPS_Override : BOOL := FALSE;
    {attribute 'pytmc' := 'pv: CRIX:DPL:MMS:X:EPS:OVRD_COUNTDOWN'}
    tEPS_TimerCountDown : STRING := TIME_TO_STRING(T#0s);
    fbResetTimer : FB_RestTimer;

    bInit 		: BOOL := TRUE;
    bFullRange 	: BOOL;

    fbEPS		: FB_EPS;
    fbCheckEPS 	: FB_CheckEPS;

END_VAR

IF bInit THEN
    // Set Inital Values
    aDPL_X_EPS[1].fBwd_Limits := 10;
    aDPL_X_EPS[1].fFwd_Limits := 80;

    aDPL_X_EPS[2].fBwd_Limits := 10;
    aDPL_X_EPS[2].fFwd_Limits := 30;

    //aDPL_X_EPS[3].fBwd_Limits := 60;
    aDPL_X_EPS[3].fFwd_Limits := 80;

    bInit := FALSE;
END_IF

aDPL_X_EPS[3].fBwd_Limits := fOBJ_X + 30;

fbEPS(eps:=aDPL_X_EPS[2].stEPS);
fbEPS.setMessage('SDS_RX in [124, 215');
fbEPS.setBit(0, F_InRange(fSDS_RX, 124, 215));

fbEPS(eps:=aDPL_X_EPS[3].stEPS);
fbEPS.setMessage('DPL_Z in [-10, 30]');
fbEPS.setBit(0, F_InRange(fDPL_Z, -10, 30));

bFullRange := (NOT aDPL_X_EPS[2].stEPS.bEPS_OK) AND (NOT aDPL_X_EPS[3].stEPS.bEPS_OK);

fbEPS(eps:=aDPL_X_EPS[1].stEPS);
fbEPS.setMessage('Full Range');
fbEPS.setBit(0, bFullRange);

fbResetTimer(bInput:=bEPS_Override, tElapseTime:=tEPS_OVRD_RESET_TIME, tCountDown:=tEPS_TimerCountDown);
fbCheckEPS(stMotor:= M1, fPosition:=fDPL_X, aEPSLimits:= aDPL_X_EPS, stForwardMotorEPS:=M1.stEPSForwardEnable, stBackwardMotorEPS:= M1.stEPSBackwardEnable, bEPS_Override:=bEPS_Override);

END_PROGRAM

// ---- POUs/EPS/InjectorMotorEPSLimits/PRG_DPL_Y_EPS.TcPOU
PROGRAM PRG_DPL_Y_EPS
VAR
    {attribute 'pytmc' := 'pv: CRIX:DPL:MMS:Y:EPS'}
    aDPL_Y_EPS		: ARRAY [1 .. 2] OF ST_EPSLimits;

    {attribute 'pytmc' := 'pv: CRIX:DPL:MMS:Y:EPS:OVRD_MODE'}
    bEPS_Override : BOOL := FALSE;
    {attribute 'pytmc' := 'pv: CRIX:DPL:MMS:Y:EPS:OVRD_COUNTDOWN'}
    tEPS_TimerCountDown : STRING := TIME_TO_STRING(T#0s);
    fbResetTimer : FB_RestTimer;

    bInit 		: BOOL := TRUE;
    bFullRange	: BOOL;

       fbEPS		: FB_EPS;
    fbCheckEPS 	: FB_CheckEPS;
END_VAR

IF bInit THEN
    // Set Inital Values
    aDPL_Y_EPS[1].fBwd_Limits := -1;
    aDPL_Y_EPS[1].fFwd_Limits := 80;

    aDPL_Y_EPS[2].fBwd_Limits := 40;
    aDPL_Y_EPS[2].fFwd_Limits := 80;

    bInit := FALSE;
END_IF

fbEPS(eps:=aDPL_Y_EPS[2].stEPS);
fbEPS.setMessage('DPL_Z in [-10,30];RCC in [-11,11]');
fbEPS.setBit(0, F_InRange(fDPL_Z, -10, 30));
fbEPS.setBit(1, F_InRange(fRCC_Z, -11, 11));

bFullRange := NOT aDPL_Y_EPS[2].stEPS.bEPS_OK;

fbEPS(eps:=aDPL_Y_EPS[1].stEPS);
fbEPS.setMessage('Full Range');
fbEPS.setBit(0, bFullRange);

fbResetTimer(bInput:=bEPS_Override, tElapseTime:=tEPS_OVRD_RESET_TIME, tCountDown:=tEPS_TimerCountDown);
fbCheckEPS(stMotor:=M2, fPosition:=M2.stAxisStatus.fActPosition, aEPSLimits:=aDPL_Y_EPS, stForwardMotorEPS:=M2.stEPSForwardEnable, stBackwardMotorEPS:= M2.stEPSBackwardEnable, bEPS_Override:= bEPS_Override);

END_PROGRAM

// ---- POUs/EPS/InjectorMotorEPSLimits/PRG_DPL_Z_EPS.TcPOU
PROGRAM PRG_DPL_Z_EPS
VAR
    {attribute 'pytmc' := 'pv: CRIX:DPL:MMS:Z:EPS'}
    aDPL_Z_EPS 	    : ARRAY [1 .. 4] OF ST_EPSLimits;

    {attribute 'pytmc' := 'pv: CRIX:DPL:MMS:Z:EPS:OVRD_MODE'}
    bEPS_Override: BOOL := FALSE;
    {attribute 'pytmc' := 'pv: CRIX:DPL:MMS:Z:EPS:OVRD_COUNTDOWN'}
    tEPS_TimerCountDown : STRING := TIME_TO_STRING(T#0s);
    fbResetTimer : FB_RestTimer;

    bInit 		: BOOL := TRUE;
    bFullRange 	: BOOL;

    fbEPS		: FB_EPS;
    fbCheckEPS 	: FB_CheckEPS;
END_VAR

IF bInit THEN
    // Set Inital Values
    aDPL_Z_EPS[1].fBwd_Limits := -10;
    aDPL_Z_EPS[1].fFwd_Limits := 100;

    aDPL_Z_EPS[2].fBwd_Limits := 30;
    aDPL_Z_EPS[2].fFwd_Limits := 100;

    aDPL_Z_EPS[3].fBwd_Limits := 30;
    aDPL_Z_EPS[3].fFwd_Limits := 100;

    aDPL_Z_EPS[4].fBwd_Limits := 30;
    aDPL_Z_EPS[4].fFwd_Limits := 100;

    bInit := FALSE;
END_IF

fbEPS(eps:=aDPL_Z_EPS[2].stEPS);
fbEPS.setMessage('DPL X in [10, OBJ_X + 30]');
fbEPS.setBit(0, F_InRange(fDPL_X, 10, fOBJ_X + 30));

fbEPS(eps:=aDPL_Z_EPS[3].stEPS);
fbEPS.setMessage('RCC Y in [-34,10];RCC_Z in [-11,11]');
fbEPS.setBit(0, F_InRange(fRCC_Y, -34, 10));
fbEPS.setBit(1, F_InRange(fRCC_Z, -11, 11));

fbEPS(eps:=aDPL_Z_EPS[4].stEPS);
fbEPS.setMessage('RCC_Y in [-38,-34];RCC_Z in [-11,11];DPL_Y in [-1,40]');
fbEPS.setBit(0, F_InRange(fRCC_Y, -38, -34));
fbEPS.setBit(1, F_InRange(fRCC_Z, -11, 11));
fbEPS.setBit(2, F_InRange(fDPL_Y, -1, 40));

bFullRange := (NOT aDPL_Z_EPS[2].stEPS.bEPS_OK) AND (NOT aDPL_Z_EPS[3].stEPS.bEPS_OK) AND (NOT aDPL_Z_EPS[4].stEPS.bEPS_OK);

fbEPS(eps:=aDPL_Z_EPS[1].stEPS);
fbEPS.setMessage('Full Range');
fbEPS.setBit(0, bFullRange);

fbResetTimer(bInput:=bEPS_Override, tElapseTime:=tEPS_OVRD_RESET_TIME, tCountDown:=tEPS_TimerCountDown);
fbCheckEPS(stMotor:=M3, fPosition:=fDPL_Z, aEPSLimits:= aDPL_Z_EPS, stForwardMotorEPS:=M3.stEPSForwardEnable, stBackwardMotorEPS:= M3.stEPSBackwardEnable, bEPS_Override:=bEPS_Override);

END_PROGRAM

// ---- POUs/EPS/InjectorMotorEPSLimits/PRG_EPS.TcPOU
PROGRAM PRG_EPS
VAR
END_VAR

// Update Motor Positions before Using them in EPS Checks
fDPL_X  := M1.stAxisStatus.fActPosition;

fSDS_RX 	:= M19.stAxisStatus.fActPosition;
fSDS_Y      := M17.stAxisStatus.fActPosition;
fSDS_Z_ENC  := M36.stAxisStatus.fActPosition;

fDPL_Z 		:= M3.stAxisStatus.fActPosition;
fDPL_Y 		:= M2.stAxisStatus.fActPosition;

fRCC_Z 		:= M39.stAxisStatus.fActPosition;
fRCC_Y 		:= M38.stAxisStatus.fActPosition;

fOBJ_X		:= M4.stAxisStatus.fActPosition;

PRG_SDS_Y_EPS();
PRG_SDS_RX_EPS();
PRG_SDS_ZENCODER_EPS();

PRG_DPL_X_EPS();
PRG_DPL_Y_EPS();
PRG_DPL_Z_EPS();

PRG_RCC_Y_EPS();
PRG_RCC_Z_EPS();

PRG_OBJ_X_EPS();

END_PROGRAM

// ---- POUs/EPS/InjectorMotorEPSLimits/PRG_SDS_Y_EPS.TcPOU
PROGRAM PRG_SDS_Y_EPS
VAR
    {attribute 'pytmc' := 'pv: CRIX:SDS:MMS:Y:EPS'}
    aSDS_Y_EPS 		: ARRAY [1 .. 5] OF ST_EPSLimits;

    {attribute 'pytmc' := 'pv: CRIX:SDS:MMS:Y:EPS:OVRD_MODE'}
    bEPS_Override : BOOL := FALSE;

    {attribute 'pytmc' := 'pv: CRIX:SDS:MMS:Y:EPS:OVRD_COUNTDOWN'}
    tEPS_TimerCountDown : STRING := TIME_TO_STRING(T#0s);
    fbResetTimer : FB_RestTimer;

    bInit 		: BOOL := TRUE;
    bFullRange	: BOOL;
    nIndex 		: uint;
    nEPSIndex 	: uint;

    fbEPS		: FB_EPS;;
    fbCheckEPS 	: FB_CheckEPS;
END_VAR

// SDS Y EPS
IF bInit THEN
    // Set Inital Values
    aSDS_Y_EPS[1].fBwd_Limits := 20;
    aSDS_Y_EPS[1].fFwd_Limits := 45;

    aSDS_Y_EPS[2].fBwd_Limits := 37.5;
    aSDS_Y_EPS[2].fFwd_Limits := 38.5;

    aSDS_Y_EPS[3].fBwd_Limits := 30;
    aSDS_Y_EPS[3].fFwd_Limits := 38.5;

    aSDS_Y_EPS[4].fBwd_Limits := 30;
    aSDS_Y_EPS[4].fFwd_Limits := 38.5;

    aSDS_Y_EPS[5].fBwd_Limits := 30;
    aSDS_Y_EPS[5].fFwd_Limits := 45;


    bInit := FALSE;
END_IF

// Set EPS conditions
fbEPS(eps:= aSDS_Y_EPS[2].stEPS);
fbEPS.setMessage('SDS_Z_ENC in [-1,3.05]');
fbEPS.setBit(0, F_InRange(fSDS_Z_ENC, -1, 3.05));

fbEPS(eps:= aSDS_Y_EPS[3].stEPS);
fbEPS.setMessage('SDS_Z_ENC in [3.05, 3.4];SDS_RX in [215, 220]');
fbEPS.setBit(0, F_InRange(fSDS_Z_ENC, 3.05, 3.4));
fbEPS.setBit(1, F_InRange(fSDS_RX, 215, 220));

fbEPS(eps:= aSDS_Y_EPS[4].stEPS);
fbEPS.setMessage('SDS_Z_ENC in [3.05, 3.8];SDS_RX in [124, 215]');
fbEPS.setBit(0, F_InRange(fSDS_Z_ENC, 3.05, 3.8));
fbEPS.setBit(1, F_InRange(fSDS_RX, 124, 215));

fbEPS(eps:= aSDS_Y_EPS[5].stEPS);
fbEPS.setDescription('SDS_Z_ENC in [3.8, 4];(SDS_Y - RCC) <= nozzle_catcher_offset');
fbEPS.setBit(0, F_InRange(fSDS_Z_ENC, 3.8, 4));
fbEPS.setBit(1, (fSDS_Y - fRCC_Y) <= fNozzleCatcherOffset);

aSDS_Y_EPS[5].fBwd_Limits := fNozzleCatcherOffset + fRCC_Y;


bFullRange := (NOT aSDS_Y_EPS[2].stEPS.bEPS_OK) AND (NOT aSDS_Y_EPS[3].stEPS.bEPS_OK) AND(NOT aSDS_Y_EPS[4].stEPS.bEPS_OK) AND (NOT aSDS_Y_EPS[5].stEPS.bEPS_OK);
fbEPS(eps:= aSDS_Y_EPS[1].stEPS);
fbEPS.setDescription('Full Range');
fbEPS.setBit(0, bFullRange); // FULL RANGE


fbResetTimer(bInput:=bEPS_Override, tElapseTime:=tEPS_OVRD_RESET_TIME, tCountDown:=tEPS_TimerCountDown);
fbCheckEPS(stMotor:=M17, fPosition:=fSDS_Y, aEPSLimits:=aSDS_Y_EPS, stForwardMotorEPS:=M17.stEPSForwardEnable, stBackwardMotorEPS:= M17.stEPSBackwardEnable, bEPS_Override:=bEPS_Override);

END_PROGRAM

// ---- POUs/EPS/InjectorMotorEPSLimits/PRG_SDS_RX_EPS.TcPOU
PROGRAM PRG_SDS_RX_EPS
VAR
    {attribute 'pytmc' := 'pv: CRIX:SDS:MMS:RX:EPS'}
    aSDS_RX_EPS 	: ARRAY [1 .. 5] OF ST_EPSLimits;

    {attribute 'pytmc' := 'pv: CRIX:SDS:MMS:RX:EPS:OVRD_MODE'}
    bEPS_Override : BOOL := FALSE;

    {attribute 'pytmc' := 'pv: CRIX:SDS:MMS:RX:EPS:OVRD_COUNTDOWN'}
    tEPS_TimerCountDown : STRING := TIME_TO_STRING(T#0s);
    fbResetTimer : FB_RestTimer;

    bInit 		: BOOL := TRUE;

    bSDS_RX_FullRange : BOOL;

    fbEPS		: FB_EPS;
    fbCheckEPS 	: FB_CheckEPS;

END_VAR

IF bInit THEN
    // Set Inital Values
    aSDS_RX_EPS[1].fBwd_Limits := 124;
    aSDS_RX_EPS[1].fFwd_Limits := 218;

    aSDS_RX_EPS[2].fBwd_Limits := 215;
    aSDS_RX_EPS[2].fFwd_Limits := 218;

    aSDS_RX_EPS[3].fBwd_Limits := 215;
    aSDS_RX_EPS[3].fFwd_Limits := 218;

    aSDS_RX_EPS[4].fBwd_Limits := 124;
    aSDS_RX_EPS[4].fFwd_Limits := 134;

    aSDS_RX_EPS[5].fBwd_Limits := 124;
    aSDS_RX_EPS[5].fFwd_Limits := 134;

    bInit := FALSE;
END_IF

// Set EPS conditions
fbEPS(eps:=aSDS_RX_EPS[1].stEPS);
fbEPS.setMessage('SDS_Z_ENC in [3.05,3.4];SDS_Y in [30,38.5];RCC_Y in [-38,-34];DPL_X in [10,30]');
fbEPS.setBit(0, F_InRange(fSDS_Z_ENC, -1 , 3.4));
fbEPS.setBit(1, F_InRange(fSDS_Y, 30, 38.5));
fbEPS.setBit(2, F_InRange(fRCC_Y, -38, -34));
fbEPS.setBit(3, F_InRange(fDPL_X, 10, 30));

bSDS_RX_FullRange := aSDS_RX_EPS[1].stEPS.bEPS_OK; // FULL RANGE CONDITION

fbEPS(eps:=aSDS_RX_EPS[2].stEPS);
fbEPS.setMessage('SDS_Z_ENC in [-1, 3.05]');
fbEPS.setBit(0, F_InRange(fSDS_Z_ENC, -1.0, 3.05));
fbEPS.setBit(1, NOT bSDS_RX_FullRange); // NOT FULL RANGE COND.

fbEPS(eps:=aSDS_RX_EPS[3].stEPS);
fbEPS.setMessage('SDS_Z_ENC in [3.05, 3.4];SDS_RX in [215, 220];Not Full Range');
fbEPS.setBit(0, F_InRange(fSDS_Z_ENC, 3.05, 3.4));
fbEPS.setBit(1, F_InRange(fSDS_RX, 215, 220));
fbEPS.setBit(2, NOT bSDS_RX_FullRange); // NOT FULL RANGE COND.

fbEPS(eps:=aSDS_RX_EPS[4].stEPS);
fbEPS.setMessage('SDS_Z_ENC in [3.4, 4]');
fbEPS.setBit(0, F_InRange(fSDS_Z_ENC, 3.4, 4));

fbEPS(eps:=aSDS_RX_EPS[5].stEPS);
fbEPS.setMessage('SDS_Z_ENC in [3.05,3.4];SDS_RX in [124, 134];Not Full Range');
fbEPS.setBit(0, F_InRange(fSDS_Z_ENC, 3.05, 3.4));
fbEPS.setBit(1, F_InRange(fSDS_RX, 124, 134));
fbEPS.setBit(2, NOT bSDS_RX_FullRange); // NOT FULL RANGE COND.

fbResetTimer(bInput:=bEPS_Override, tElapseTime:=tEPS_OVRD_RESET_TIME, tCountDown:=tEPS_TimerCountDown);
fbCheckEPS(stMotor:=M19, fPosition:= fSDS_RX, aEPSLimits:= aSDS_RX_EPS, stForwardMotorEPS:=M19.stEPSForwardEnable, stBackwardMotorEPS:= M19.stEPSBackwardEnable, bEPS_Override:=bEPS_Override);

END_PROGRAM

// ---- POUs/EPS/InjectorMotorEPSLimits/PRG_SDS_ZENCODER_EPS.TcPOU
PROGRAM PRG_SDS_ZENCODER_EPS
VAR
    {attribute 'pytmc' := 'pv: CRIX:SDS:MMS:ZENC:EPS'}
    aSDS_Z_ENC_EPS	: ARRAY [1 .. 5] OF ST_EPSLimits;

    {attribute 'pytmc' := 'pv: CRIX:SDS:MMS:ZENC:EPS:OVRD_MODE'}
    bEPS_Override : BOOL := FALSE;

    {attribute 'pytmc' := 'pv: CRIX:SDS:MMS:ZENC:EPS:OVRD_COUNTDOWN'}
    tEPS_TimerCountDown : STRING := TIME_TO_STRING(T#0s);
    fbResetTimer : FB_RestTimer;

    bInit       : BOOL := TRUE;
    bSDS_vert_transport_state : BOOL;
    bFullRange	: BOOL;
    bUnknownState	: BOOL;

    fbEPS		: FB_EPS;
    fbCheckEPS 	: FB_CheckEPS;
END_VAR

IF bInit THEN

    aSDS_Z_ENC_EPS[1].fBwd_Limits := -1;
    aSDS_Z_ENC_EPS[1].fFwd_Limits := 3.4;

    aSDS_Z_ENC_EPS[2].fBwd_Limits := 3.05;
    aSDS_Z_ENC_EPS[2].fFwd_Limits := 3.4;

    aSDS_Z_ENC_EPS[3].fBwd_Limits := 3.05;
    aSDS_Z_ENC_EPS[3].fFwd_Limits := 3.4;

    aSDS_Z_ENC_EPS[4].fBwd_Limits := 3.05;
    aSDS_Z_ENC_EPS[4].fFwd_Limits := 4;

    aSDS_Z_ENC_EPS[5].fBwd_Limits := 3.8;
    aSDS_Z_ENC_EPS[5].fFwd_Limits := 4;

    bInit := FALSE;
END_IF


bSDS_vert_transport_state := F_InRange(fSDS_Y, 30, 38.5) AND F_InRange(fSDS_RX, 124, 134) AND (fDPL_X < 30) AND (fRCC_Y < -34);

fbEPS(eps:=aSDS_Z_ENC_EPS[1].stEPS);
fbEPS.setMessage('SDS_RX in [215, 220];SDS_Y in [37.5, 38.5]');
fbEPS.setBit(0, F_InRange(fSDS_RX, 215, 220));
fbEPS.setBit(1, F_InRange(fSDS_Y, 37.5, 38.5));

fbEPS(eps:=aSDS_Z_ENC_EPS[2].stEPS);
fbEPS.setMessage('SDS_RX in [134, 220];SDS_Y in [30, 38.5]');
fbEPS.setBit(0, F_InRange(fSDS_RX, 134, 220));
fbEPS.setBit(1, F_InRange(fSDS_Y, 30, 37.5));

fbEPS(eps:=aSDS_Z_ENC_EPS[3].stEPS);
fbEPS.setMessage('SDS_RX in [124, 134];SDS_Z_ENC in [3.05, 3.45];NOT SDS VERT. TRANSPORT STATE');
fbEPS.setBit(0, F_InRange(fSDS_RX, 124, 134));
fbEPS.setBit(1, F_InRange(fSDS_Z_ENC, 3.05, 3.45));
fbEPS.setBit(2, NOT bSDS_vert_transport_state); // NOT INJECTOR Vertical Tansport Condition

fbEPS(eps:=aSDS_Z_ENC_EPS[4].stEPS);
fbEPS.setMessage('SDS_RX in [124, 134];SDS_Y in [30, 38.5];RCC_Y in [-38,-34];DPL_X in [10,30]');
fbEPS.setBit(0, F_InRange(fSDS_RX, 124, 134));
fbEPS.setBit(1, F_InRange(fSDS_Y, 30, 38.5));
fbEPS.setBit(2, F_InRange(fRCC_Y, -38, -34));
fbEPS.setBit(3, F_InRange(fDPL_X, 10, 30));

fbEPS(eps:=aSDS_Z_ENC_EPS[5].stEPS);
fbEPS.setMessage('SDS_RX in [124, 134];SDS_Z_ENC in [3.75, 4]; NOT SDS VERT. TRANSPORT State');
fbEPS.setBit(0, F_InRange(fSDS_RX, 124, 134));
fbEPS.setBit(1, F_InRange(fSDS_Z_ENC, 3.75, 4));
fbEPS.setBit(2, NOT bSDS_vert_transport_state); // NOT INJECTOR Vertical Transport Condition


fbResetTimer(bInput:=bEPS_Override, tElapseTime:=tEPS_OVRD_RESET_TIME, tCountDown:=tEPS_TimerCountDown);
fbCheckEPS(stMotor:=M18, fPosition:=fSDS_Z_ENC, stForwardMotorEPS:= M18.stEPSBackwardEnable, stBackwardMotorEPS:=M18.stEPSForwardEnable, aEPSLimits:=aSDS_Z_ENC_EPS, bEPS_Override:=bEPS_Override);

END_PROGRAM

// ---- POUs/EPS/InjectorMotorEPSLimits/PRG_RCC_Y_EPS.TcPOU
PROGRAM PRG_RCC_Y_EPS
VAR
    {attribute 'pytmc' := 'pv: CRIX:RCC:MMS:Y:EPS'}
    aRCC_Y_EPS 	    : ARRAY [1 .. 4] OF ST_EPSLimits;

    {attribute 'pytmc' := 'pv: CRIX:RCC:MMS:Y:EPS:OVRD_MODE'}
    bEPS_Override : BOOL :=  FALSE;

    {attribute 'pytmc' := 'pv: CRIX:RCC:MMS:Y:EPS:OVRD_COUNTDOWN'}
    tEPS_TimerCountDown : STRING := TIME_TO_STRING(T#0s);
    fbResetTimer : FB_RestTimer;

    bInit 		: BOOL := TRUE;
    bFullRange	: BOOL;

    fbEPS		: FB_EPS;
    fbCheckEPS 	: FB_CheckEPS;
END_VAR

 IF bInit THEN
    // Set Inital Values
    aRCC_Y_EPS[1].fBwd_Limits := -38;
    aRCC_Y_EPS[1].fFwd_Limits := 10;

    aRCC_Y_EPS[2].fBwd_Limits := -38;
    aRCC_Y_EPS[2].fFwd_Limits := -34;

    aRCC_Y_EPS[3].fBwd_Limits := -38;
    aRCC_Y_EPS[3].fFwd_Limits := -34;

    aRCC_Y_EPS[4].fBwd_Limits := -38;
    aRCC_Y_EPS[4].fFwd_Limits := 0; // VARIBLE

    bInit := FALSE;
END_IF

fbEPS(eps:=aRCC_Y_EPS[2].stEPS);
fbEPS.setMessage('SDS_RX in [124, 215];SDS_Z_ENC in [3.05, 3.8]');
fbEPS.setBit(0, F_InRange(fSDS_RX, 124, 215));
fbEPS.setBit(1, F_InRange(fSDS_Z_ENC, 3.05, 3.8));

fbEPS(eps:=aRCC_Y_EPS[3].stEPS);
fbEPS.setMessage('DPL_Z in [-10,30];RCC_Z in [-15,11]');
fbEPS.setBit(0, F_InRange(fDPL_Z, -10, 30));
fbEPS.setBit(1, F_InRange(fRCC_Z, -15, 11));

fbEPS(eps:=aRCC_Y_EPS[4].stEPS);
fbEPS.setMessage('SDS_Z_ENC in [3.8, 4];SDS_Y - RCC_Y <= nozzle_catcher_offset');
fbEPS.setBit(0, F_InRange(fSDS_Z_ENC, 3.8, 4));
fbEPS.setBit(1, (fSDS_Y - fRCC_Y) <= fNozzleCatcherOffset);

aRCC_Y_EPS[4].fFwd_Limits := fSDS_Y - fNozzleCatcherOffset; // Variable Limits


bFullRange := (NOT aRCC_Y_EPS[2].stEPS.bEPS_OK) AND (NOT aRCC_Y_EPS[3].stEPS.bEPS_OK) AND (NOT aRCC_Y_EPS[4].stEPS.bEPS_OK);

fbEPS(eps:=aRCC_Y_EPS[1].stEPS);
fbEPS.setMessage('Full Range');
fbEPS.setBit(0, bFullRange);

fbResetTimer(bInput:=bEPS_Override, tElapseTime:=tEPS_OVRD_RESET_TIME, tCountDown:=tEPS_TimerCountDown);
fbCheckEPS(stMotor:=M38, fPosition:=fRCC_Y, aEPSLimits:=aRCC_Y_EPS, stForwardMotorEPS:=M38.stEPSForwardEnable, stBackwardMotorEPS:= M38.stEPSBackwardEnable, bEPS_Override:=bEPS_Override);

END_PROGRAM

// ---- POUs/EPS/InjectorMotorEPSLimits/PRG_RCC_Z_EPS.TcPOU
PROGRAM PRG_RCC_Z_EPS
VAR
    {attribute 'pytmc' := 'pv: CRIX:RCC:MMS:Z:EPS'}
    aRCC_Z_EPS	    : ARRAY [1 .. 3] OF ST_EPSLimits;

    {attribute 'pytmc' := 'pv: CRIX:RCC:MMS:Z:EPS:OVRD_MODE'}
    bEPS_Override: BOOL := FALSE;

    {attribute 'pytmc' := 'pv: CRIX:RCC:MMS:Z:EPS:OVRD_COUNTDOWN'}
    tEPS_TimerCountDown : STRING := TIME_TO_STRING(T#0s);
    fbResetTimer : FB_RestTimer;
    bInit 		: BOOL := TRUE;
    bFullRange	: BOOL;

    fbEPS		: FB_EPS;
    fbCheckEPS 	: FB_CheckEPS;
END_VAR

IF bInit THEN
    // Set Inital Values
    aRCC_Z_EPS[1].fBwd_Limits := -18;
    aRCC_Z_EPS[1].fFwd_Limits := 11;

    aRCC_Z_EPS[2].fBwd_Limits := -18;
    aRCC_Z_EPS[2].fFwd_Limits := -11;

    aRCC_Z_EPS[3].fBwd_Limits := -18;
    aRCC_Z_EPS[3].fFwd_Limits := -11;

    bInit := FALSE;
END_IF


fbEPS(eps:=aRCC_Z_EPS[2].stEPS);
fbEPS.setMessage('DPL_Z in [-10,30];DPL_Y in [-1,40]');
fbEPS.setBit(0, F_InRange(fDPL_Z, -10, 30));
fbEPS.setBit(1, F_InRange(fDPL_Y, -1, 40));

fbEPS(eps:=aRCC_Z_EPS[3].stEPS);
fbEPS.setMessage('DPL_Z in [-10, 30];RCC_Y in [-34,10]');
fbEPS.setBit(0, F_InRange(fDPL_Z, -10, 30));
fbEPS.setBit(1, F_InRange(fRCC_Y, -34, 10));

bFullRange := (NOT aRCC_Z_EPS[2].stEPS.bEPS_OK) AND (NOT aRCC_Z_EPS[3].stEPS.bEPS_OK);

fbEPS(eps:=aRCC_Z_EPS[1].stEPS);
fbEPS.setMessage('Full Range');
fbEPS.setBit(0, bFullRange);

fbResetTimer(bInput:=bEPS_Override, tElapseTime:=tEPS_OVRD_RESET_TIME, tCountDown:= tEPS_TimerCountDown);
fbCheckEPS(stMotor:= M39, fPosition:=fRCC_Z, aEPSLimits:=aRCC_Z_EPS, stForwardMotorEPS:=M39.stEPSForwardEnable, stBackwardMotorEPS:= M39.stEPSBackwardEnable, bEPS_Override:=bEPS_Override);

END_PROGRAM

// ---- POUs/EPS/InjectorMotorEPSLimits/PRG_OBJ_X_EPS.TcPOU
PROGRAM PRG_OBJ_X_EPS
VAR
    {attribute 'pytmc' := 'pv: CRIX:OBJ:MMS:X:EPS'}
    aOBJ_X_EPS 	    : ARRAY [1 .. 2] OF ST_EPSLimits;

    {attribute 'pytmc' := 'pv: CRIX:OBJ:MMS:X:EPS:OVRD_MODE'}
    bEPS_Override: BOOL := FALSE;
    {attribute 'pytmc' := 'pv: CRIX:OBJ:MMS:X:EPS:OVRD_COUNTDOWN'}
    tEPS_TimerCountDown : STRING := TIME_TO_STRING(T#0s);
    fbResetTimer : FB_RestTimer;

    bInit 		: BOOL := TRUE;
    bFullRange 	: BOOL;

    fbEPS		: FB_EPS;
    fbCheckEPS 	: FB_CheckEPS;
END_VAR

IF bInit THEN
    // Set Inital Values
    aOBJ_X_EPS[1].fBwd_Limits := -2;
    aOBJ_X_EPS[1].fFwd_Limits := 32;

    aOBJ_X_EPS[2].fBwd_Limits := -2;

    bInit := FALSE;
END_IF

aOBJ_X_EPS[2].fFwd_Limits := MIN(fDPL_X - 30, 32);

fbEPS(eps:=aOBJ_X_EPS[2].stEPS);
fbEPS.setMessage('DPL Z in [10, 30]');
fbEPS.setBit(0, F_InRange(fDPL_Z, -10, 30));

bFullRange := (NOT aOBJ_X_EPS[2].stEPS.bEPS_OK);

fbEPS(eps:=aOBJ_X_EPS[1].stEPS);
fbEPS.setMessage('Full Range');
fbEPS.setBit(0, bFullRange);


fbResetTimer(bInput:=bEPS_Override, tElapseTime:=tEPS_OVRD_RESET_TIME, tCountDown:=tEPS_TimerCountDown);
fbCheckEPS(stMotor:=M4, fPosition:=fOBJ_X, aEPSLimits:= aOBJ_X_EPS, stForwardMotorEPS:=M4.stEPSForwardEnable, stBackwardMotorEPS:= M4.stEPSBackwardEnable, bEPS_Override:=bEPS_Override);

END_PROGRAM

// ---- POUs/PRG_Main.TcPOU
PROGRAM PRG_Main
VAR
    //stTestMotor1	:	DUT_SimMotor;
    //fbTestMotor		:	FB_SIM_MOTOR;
    bInit			:	BOOL := FALSE;
    DPState : INT;
    arrStates : ARRAY [1..9] OF ENUM_DiagPaddle;
    bDPaddleOK : BOOL;

END_VAR

IF NOT bInit THEN
    bInit := TRUE;
END_IF

// Add interlock logic to this later
bDPaddleOK := TRUE;
//PRG_DiagnosticPaddle(xMoveOK:=bDPaddleOK);

//PRG_QueueTest();

//PRG_Test_AdjacentStates();

//PRG_BFS();

PRG_EPS();
PRG_DiagnosticPaddleMotors();

PRG_QuestarMotors();

PRG_PointDetectorMotors();

PRG_CryoStat();
PRG_RCI();
PRG_Camera();
PRG_FZP();
PRG_ObjectivesMotors();
PRG_RCC();
PRG_VLS();
PRG_InjectorMotors();
PRG_Illumination();
PRG_CryoPump();
PRG_FiberLite();

PRG_PMPS();

END_PROGRAM
